PROGRAM MAIN
VAR
END_VAR

P_ModeControl();

END_PROGRAM

(* stored: Version 1.1.0.1, ProductVersion 3.1.4024.12
   POU MAIN: Id {2bc9bab6-929f-4cb7-be61-76e5b0d42c48}, SpecialFunc None *)
